TYPE ST_WidgetData :
STRUCT
	{attribute 'iot.NestedStructIcon' := 'Floor'}
	{attribute 'iot.DisplayName' := 'All Widgets Overview'}
	stWidgetsOverview	: ST_Widgets_Overview;
	
	{attribute 'iot.NestedStructIcon' := 'Lightbulb'}
	{attribute 'iot.DisplayName' := 'Light Widgets'}
	stLights		: ST_Widgets_Lightings;
	
	{attribute 'iot.NestedStructIcon' := 'Blinds'}
	{attribute 'iot.DisplayName' := 'Blinds Widgets'}
	stBlinds		: ST_Widgets_Blinds;
	
	{attribute 'iot.NestedStructIcon' := 'Plug'}
	{attribute 'iot.DisplayName' := 'Plug Widgets'}
	stPlugs			: ST_Widgets_Plugs;
	
	{attribute 'iot.NestedStructIcon' := 'Temperature'}
	{attribute 'iot.DisplayName' := 'AC Widgets'}
	stAC			: ST_Widgets_AC;
	
	{attribute 'iot.NestedStructIcon' := 'Co2'}
	{attribute 'iot.DisplayName' := 'Ventilation Widgets'}
	stVentilation	: ST_Widgets_Ventilation;
	
	{attribute 'iot.NestedStructIcon' := 'Clock'}
	{attribute 'iot.DisplayName' := 'Time Switch Widgets'}
	stTimeSwitch	: ST_Widgets_TimeSwitch;
	
	{attribute 'iot.NestedStructIcon' := 'Room'}
	{attribute 'iot.DisplayName' := 'General Widgets'}
	stGeneral		: ST_Widgets_GeneralWidget;
END_STRUCT
END_TYPE

(* stored: Version 1.1.0.1, ProductVersion 3.1.4024.11
   DUT ST_WidgetData: Id {499993c7-8b57-486e-9379-8d02e8d3f92e} *)
